DATA_BLOCK "dbArchiveAutoEom"
{ S7_Optimized_Access := 'TRUE' }
VERSION : 0.8
NON_RETAIN
"fbArchiveAutoEom"

BEGIN

END_DATA_BLOCK

